PROGRAM MQTTCOMM
VAR
    fbMqttClient    :FB_IotMqttClient;
    bSetParameter   :BOOL 		 	:= TRUE;
    bConnect        :BOOL 		 	:= TRUE;	
	
	(* published message *)
	
	MotionStatusPub :STRING(255)	:= 'MOTION/STATUS';
	MotionCTREcho	:STRING(255)	:= 'MOTION/CTR_ECHO';
	MotionINSTREcho	:STRING(255)	:= 'MOTION/INSTR_ECHO';
	HBEcho			:STRING(255)	:= 'MOTION/HB_ECHO';

	ScriptSend		:STRING(255)	:= 'MOTION/SCRIPTSEND';
	ScriptNames		:STRING(255)	:= 'MOTION/SCRIPTNAMES';
	sPayloadPub 	:STRING(1000);
	fbTimer 		:TON			:= (PT:=T#500MS);
	HBtimer 		:TON			:= (PT:=T#1S);
	scriptTimer		:TON			:= (PT:=T#2MS);
	found 			:UDINT;	
	notreset		:BOOL			:= FALSE;
	HBcase			:INT			:= 0;
	
   (* received message *)
    SubMCTR		    :BOOL;
	SubIBuff		:BOOL;
    SubHB			:BOOL;
    {attribute 'TcEncoding':='UTF-8'}
    sTopicRcv       :STRING(255);
    {attribute 'TcEncoding':='UTF-8'}
    sPayloadRcv     :STRING(2000);
    fbMessageQueue  :FB_IotMqttMessageQueue;
    fbMessage       :FB_IotMqttMessage;	
	
	(* JSON *)
	fbJson 			:FB_JsonSaxWriter;
	fbJsonDataType 	:FB_JsonReadWriteDataType;
	fbJsonSaxReader	:FB_JsonSaxReader;
	pJsonParse		:JsonSaxHandler;
	jsonDoc    		:SJsonValue;
  	jsonProp   		:SJsonValue;
	
	ok				:BOOL;
	error			:HRESULT;
	index			:INT			:= 0;
	payload			:T_MaxString;
	scriptcnt		:INT			:= 0;
END_VAR

//takes any INT as UDINT?
//received (and echoed) messages:
//GVL_MOTION.EXT_CTR
//GVL_MOTION.InstructionBuffer
//published messages:
//GVL_MOTION.STATUS
//receive 
//GVL_MOTION.HB.HEARTBEAT

IF bSetParameter THEN
    bSetParameter								:= FALSE;
    fbMqttClient.sHostName						:= '127.0.0.1';
    fbMqttClient.nHostPort						:= 1883;
    fbMqttClient.ipMessageQueue					:= fbMessageQueue;
END_IF

fbMqttClient.Execute(bConnect);

IF fbMessageQueue.nQueuedMessages > 0 THEN
    IF fbMessageQueue.Dequeue(fbMessage:=fbMessage) THEN
        fbMessage.GetTopic(pTopic:=ADR(GVL_MOTION.TopicRcv), nTopicSize:=SIZEOF(GVL_MOTION.TopicRcv) );
        fbMessage.GetPayload(pPayload:=ADR(sPayloadRcv), nPayloadSize:=SIZEOF(sPayloadRcv), bSetNullTermination:=FALSE);
		fbJsonSaxReader.Parse(sJson := sPayloadRcv, ipHdl := pJsonParse);
		
    END_IF
END_IF

IF fbMqttClient.bConnected THEN
    IF NOT SubMCTR THEN
        SubMCTR := fbMqttClient.Subscribe(sTopic:='MOTION/CTR', eQoS:=TcIotMqttQos.AtMostOnceDelivery);
    END_IF
    IF NOT SubIBuff THEN
        SubIBuff := fbMqttClient.Subscribe(sTopic:='MOTION/INSTR_BUFFER', eQoS:=TcIotMqttQos.AtMostOnceDelivery);
    END_IF	
	IF NOT SubHB THEN
        SubHB := fbMqttClient.Subscribe(sTopic:='MOTION/HB', eQoS:=TcIotMqttQos.AtMostOnceDelivery);
    END_IF	
    fbTimer(IN:=TRUE);
	//wait for trigger from daqtask - instantaneous data ready to transmit
// 	IF GVL_DAQ.DREADY THEN
// 		GVL_DAQ.DREADY			:= FALSE;
// 		fbJson.ResetDocument();
// 		fbJson.StartObject();	
// 		fbJsonDataType.AddJsonKeyValueFromSymbol(fbJson, '', 'DATA', SIZEOF(GVL_DAQ.DATA), ADR(GVL_DAQ.DATA));
// 		fbJson.EndObject();
// 		fbJson.CopyDocument(sPayloadPub, SIZEOF(sPayLoadPub));
// 		
// 		found	:= FIND2(ADR(sPayLoadPub), ADR('}}'));
// 		DELETE2(ADR(sPayLoadPub), ADR(sPayLoadPub), SIZEOF(sPayLoadPub), 1, found + 1);
// 		DELETE2(ADR(sPayLoadPub), ADR(sPayLoadPub), SIZEOF(sPayLoadPub), 4, 1);
// 		
// 		fbMqttClient.Publish(sTopic:= DaqDataPub, pPayload:= ADR(sPayloadPub), 
// 			nPayloadSize:= LEN2(ADR(sPayloadPub)), eQoS:= TcIotMqttQos.AtMostOnceDelivery, 
// 			bRetain:= TRUE, bQueue:= FALSE );	
// 	END_IF
	
    IF fbTimer.Q THEN // publish new payload every second
		//convert xOut to JSON
        fbTimer(IN:=FALSE);
		
		fbJson.ResetDocument();
		fbJson.StartObject();
		//AddJsonValueFromSymbol does not auto format in mosquitto, this one does
		//this function doesnt work with custom data types in the struct
		//3rd variable is the struct type
		fbJsonDataType.AddJsonKeyValueFromSymbol(fbJson, '', 'STATUS', SIZEOF(GVL_MOTION.STATUS), ADR(GVL_MOTION.STATUS));
		//fbJson.AddKeyBool('EN',GVL_MOTION.xCon.Enable);
		fbJson.EndObject();
		fbJson.CopyDocument(sPayloadPub, SIZEOF(sPayLoadPub));
		
		found	:= FIND2(ADR(sPayLoadPub), ADR('}}'));
		DELETE2(ADR(sPayLoadPub), ADR(sPayLoadPub), SIZEOF(sPayLoadPub), 1, found + 1);
		DELETE2(ADR(sPayLoadPub), ADR(sPayLoadPub), SIZEOF(sPayLoadPub), 4, 1);
		
        fbMqttClient.Publish(sTopic:= MotionStatusPub, pPayload:= ADR(sPayloadPub), 
			nPayloadSize:= LEN2(ADR(sPayloadPub)), eQoS:= TcIotMqttQos.AtMostOnceDelivery, 
			bRetain:= TRUE, bQueue:= FALSE );
			
			
		fbJson.ResetDocument();
		fbJson.StartObject();
		fbJsonDataType.AddJsonKeyValueFromSymbol(fbJson, '', 'MOTION_CTR', SIZEOF(GVL_MOTION.EXT_CTR), ADR(GVL_MOTION.EXT_CTR));
		fbJson.EndObject();
		fbJson.CopyDocument(sPayloadPub, SIZEOF(sPayLoadPub));
		
		found	:= FIND2(ADR(sPayLoadPub), ADR('}}'));
		DELETE2(ADR(sPayLoadPub), ADR(sPayLoadPub), SIZEOF(sPayLoadPub), 1, found + 1);
		DELETE2(ADR(sPayLoadPub), ADR(sPayLoadPub), SIZEOF(sPayLoadPub), 4, 1);
		
		fbMqttClient.Publish(sTopic:= MotionCTREcho, pPayload:= ADR(sPayloadPub), 
			nPayloadSize:= LEN2(ADR(sPayloadPub)), eQoS:= TcIotMqttQos.AtMostOnceDelivery, 
			bRetain:= TRUE, bQueue:= FALSE );
		
		fbJson.ResetDocument();
		fbJson.StartObject();	
		fbJsonDataType.AddJsonKeyValueFromSymbol(fbJson, '', 'MOTION_INSTRUCTION', SIZEOF(GVL_MOTION.InstructionBuffer), ADR(GVL_MOTION.InstructionBuffer));
		fbJson.EndObject();
		fbJson.CopyDocument(sPayloadPub, SIZEOF(sPayLoadPub));
		
		found	:= FIND2(ADR(sPayLoadPub), ADR('}}'));
		DELETE2(ADR(sPayLoadPub), ADR(sPayLoadPub), SIZEOF(sPayLoadPub), 1, found + 1);
		DELETE2(ADR(sPayLoadPub), ADR(sPayLoadPub), SIZEOF(sPayLoadPub), 4, 1);
		
		fbMqttClient.Publish(sTopic:= MotionINSTREcho, pPayload:= ADR(sPayloadPub), 
			nPayloadSize:= LEN2(ADR(sPayloadPub)), eQoS:= TcIotMqttQos.AtMostOnceDelivery, 
			bRetain:= TRUE, bQueue:= FALSE );
	
			
		IF GVL_MOTION.LISTSTART THEN
			IF index < GVL_MOTION.LISTCNT THEN
				IF index = 0 THEN
					GVL_MOTION.SCRIPTNAME.start	:= TRUE;
				ELSIF index = (GVL_MOTION.LISTCNT - 1) THEN
					GVL_MOTION.SCRIPTNAME.end	:= TRUE; 	
				ELSE
					GVL_MOTION.SCRIPTNAME.start	:= FALSE;
					GVL_MOTION.SCRIPTNAME.end	:= FALSE;	
				END_IF
				
				GVL_MOTION.SCRIPTNAME.payload	:= GVL_MOTION.LIST[index];
				
				fbJson.ResetDocument();
				fbJson.StartObject();	
				fbJsonDataType.AddJsonKeyValueFromSymbol(fbJson, '', 'SCRIPTNAME', SIZEOF(GVL_MOTION.SCRIPTNAME), ADR(GVL_MOTION.SCRIPTNAME));
				fbJson.EndObject();
				fbJson.CopyDocument(sPayloadPub, SIZEOF(sPayLoadPub));
				
				found	:= FIND2(ADR(sPayLoadPub), ADR('}}'));
				DELETE2(ADR(sPayLoadPub), ADR(sPayLoadPub), SIZEOF(sPayLoadPub), 1, found + 1);
				DELETE2(ADR(sPayLoadPub), ADR(sPayLoadPub), SIZEOF(sPayLoadPub), 4, 1);
				
				fbMqttClient.Publish(sTopic:= ScriptNames, pPayload:= ADR(sPayloadPub), 
					nPayloadSize:= LEN2(ADR(sPayloadPub)), eQoS:= TcIotMqttQos.AtMostOnceDelivery, 
					bRetain:= TRUE, bQueue:= FALSE );	
					
				index							:= index + 1;
			ELSE
				GVL_MOTION.SCRIPTNAME.start		:= FALSE;
				GVL_MOTION.SCRIPTNAME.end		:= FALSE;
				index							:= 0;	
				GVL_MOTION.LISTSTART			:= FALSE;
				GVL_MOTION.LISTEND				:= TRUE;
			END_IF
		END_IF
    END_IF
END_IF

IF fbMqttClient.bConnected THEN
	//IF GVL_MOTION.EXT_CTR.CMDREQSCRIPT THEN
		scriptTimer(IN:=TRUE);
		IF scriptTimer.Q THEN
			scriptTimer(IN:=FALSE);
			IF scriptcnt < GVL_MOTION.STATUS.ScriptEnd THEN
				GVL_MOTION.Script[scriptcnt].index	:= scriptcnt;
				fbJson.ResetDocument();
				fbJson.StartObject();	
				fbJsonDataType.AddJsonKeyValueFromSymbol(fbJson, '', 'MOTION_INSTRUCTION', SIZEOF(GVL_MOTION.Script[scriptcnt]), ADR(GVL_MOTION.Script[scriptcnt]));
				fbJson.EndObject();
				fbJson.CopyDocument(sPayloadPub, SIZEOF(sPayLoadPub));
				
				found	:= FIND2(ADR(sPayLoadPub), ADR('}}'));
				DELETE2(ADR(sPayLoadPub), ADR(sPayLoadPub), SIZEOF(sPayLoadPub), 1, found + 1);
				DELETE2(ADR(sPayLoadPub), ADR(sPayLoadPub), SIZEOF(sPayLoadPub), 4, 1);
				
				fbMqttClient.Publish(sTopic:= ScriptSend, pPayload:= ADR(sPayloadPub), 
					nPayloadSize:= LEN2(ADR(sPayloadPub)), eQoS:= TcIotMqttQos.AtMostOnceDelivery, 
					bRetain:= TRUE, bQueue:= FALSE );
				scriptcnt						:= scriptcnt + 1;
			ELSE
				scriptcnt						:= 0;
				GVL_MOTION.EXT_CTR.CMDREQSCRIPT	:= FALSE;
			END_IF
		END_IF
	//END_IF
END_IF

IF NOT GVL_MOTION.HB.HEARTBEAT THEN
//3 second timer. set heartbeat false. control continuously sets heartbeat true, 
//after 3 cycles disable sensitive motion controls
	HBtimer(IN:=TRUE, PT := T#1S); 
ELSE
	HBtimer(IN:=FALSE);
	GVL_MOTION.HB.HEARTBEAT						:= FALSE;
END_IF	

IF HBtimer.Q THEN	
	GVL_MOTION.EXT_CTR.XJOGFW					:= FALSE;	
	GVL_MOTION.EXT_CTR.XJOGBW					:= FALSE;	
	GVL_MOTION.EXT_CTR.YJOGFW					:= FALSE;	
	GVL_MOTION.EXT_CTR.YJOGBW					:= FALSE;	
	GVL_MOTION.EXT_CTR.ZJOGFW					:= FALSE;	
	GVL_MOTION.EXT_CTR.ZJOGBW					:= FALSE;	
END_IF

END_PROGRAM

(* stored: Version 1.1.0.1, ProductVersion 3.1.4026.18
   POU MQTTCOMM: Id {6cc164ab-7114-46c3-9a99-d0016021e99e}, SpecialFunc None *)
